FUNCTION_BLOCK OperatorRelational (* Template for an empty basic function block *)
  (* Standard: 61499-2; Description: Copyright (c) 2019 Jan Holzweber This program and the accompanying materials are made available under the terms of the Eclipse Public License 2.0 which is available at https://www.eclipse.org/legal/epl-2.0/ SPDX-License-Identifier: EPL-2.0 *)
  (* Version 1.0, 2019-06-05, jholz *)
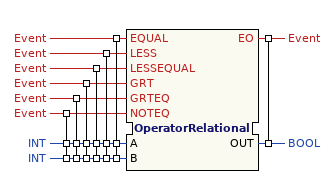
  EVENT_INPUT
    EQUAL WITH A, B;
    LESS WITH A, B;
    LESSEQUAL WITH A, B;
    GRT WITH A, B;
    GRTEQ WITH A, B;
    NOTEQ WITH A, B;
  END_EVENT
  EVENT_OUTPUT
    EO WITH OUT;
  END_EVENT
  VAR_INPUT
    A : INT;
    B : INT;
  END_VAR
  VAR_OUTPUT
    OUT : BOOL;
  END_VAR
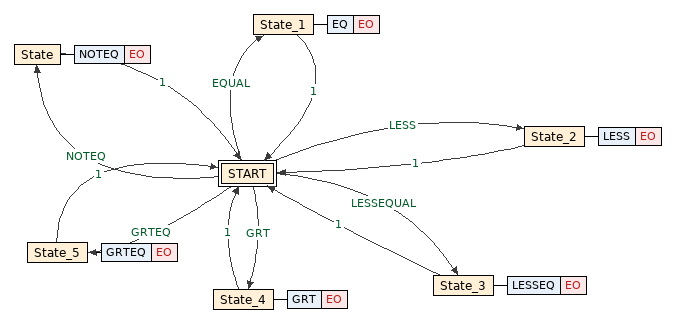
  EC_STATES
    START; (* Initial State *)
    State : NOTEQ -> EO;
    State_1 : EQ -> EO;
    State_2 : LESS -> EO;
    State_3 : LESSEQ -> EO;
    State_4 : GRT -> EO;
    State_5 : GRTEQ -> EO;
  END_STATES
  EC_TRANSITIONS
    State_1 TO START := 1;
    START TO State_1 := EQUAL;
    START TO State_2 := LESS;
    START TO State_3 := LESSEQUAL;
    START TO State_4 := GRT;
    START TO State_5 := GRTEQ;
    START TO State := NOTEQ;
    State TO START := 1;
    State_5 TO START := 1;
    State_4 TO START := 1;
    State_3 TO START := 1;
    State_2 TO START := 1;
  END_TRANSITIONS
  ALGORITHM EQ IN ST: (* new algorithm *)
OUT:=A=B;
  END_ALGORITHM
  ALGORITHM LESS IN ST: (* new algorithm *)
OUT:=A<B;
  END_ALGORITHM
  ALGORITHM LESSEQ IN ST: (* new algorithm *)
OUT:=A<=B;
  END_ALGORITHM
  ALGORITHM GRT IN ST: (* new algorithm *)
OUT:=A>B;
  END_ALGORITHM
  ALGORITHM GRTEQ IN ST: (* new algorithm *)
OUT:=A >=B;
  END_ALGORITHM
  ALGORITHM NOTEQ IN ST: (* new algorithm *)
OUT:=A <> B;
  END_ALGORITHM
END_FUNCTION_BLOCK
